(* CODESYS project Tc3_BLAKE3.library
   Company: RKe
   DefaultNamespace: Tc3_BLAKE3
   Version: 0.0.0.2
   Placeholder: Tc3_BLAKE3
   Author: Kim Robbens
   Description: Library for hash calculation with the BLAKE3 algorithm
   Title: Tc3_BLAKE3

Project tree, tasks and I/O mapping:
  libraries: Tc2_System, * (Beckhoff Automation GmbH); Tc2_Utilities, * (Beckhoff Automation GmbH); Tc3_AlgoInterfaces, * (RKe)
  DUTs/
    data type blake3_chunk_state
    data type blake3_hasher
    data type output
    data type size_t
  ITFs/
    interface IDigestBlake3: init_derive_key, init_keyed
  POUs/
    function block BLAKE3 [ST]: algorithm, chunk_state_init, chunk_state_len, chunk_state_output, chunk_state_start_flag, chunk_state_update, compress, finalize, g, hasher_add_chunk_cv, hasher_init_internal, hasher_pop_stack, hasher_push_stack, init, init_derive_key, init_keyed, key_bytes_from_hex_string, key_bytes_from_string, output_chaining_value, output_root_bytes, parent_cv, parent_output, permute, round_function, update, words_from_little_endian_bytes
  Project Information/
    function F_GetCompany [ST]
    function F_GetTitle [ST]
    function F_GetVersion [ST]
  Version/
    global variables Global_Version
  global variables ParameterList
*)

// DUTs/blake3_chunk_state
TYPE blake3_chunk_state :
STRUCT
  chaining_value				: ARRAY[0..7] OF DWORD;
  chunk_counter					: DWORD;
  block							: ARRAY[0..ParameterList.BLAKE3_BLOCK_LEN-1] OF BYTE;
  block_len						: BYTE;
  blocks_compressed				: BYTE;				
  flags							: DWORD;
END_STRUCT
END_TYPE

// DUTs/blake3_hasher
// An incremental hasher that can accept any number of writes.
TYPE blake3_hasher :
STRUCT
  chunk_state					: blake3_chunk_state;
  key_words						: ARRAY[0..7] OF DWORD;
  cv_stack 						: ARRAY[0..8*54] OF DWORD; // Space for 54 subtree chaining values:
  cv_stack_len					: BYTE;      // 2^54 * CHUNK_LEN = 2^64
  flags							: DWORD;
END_STRUCT
END_TYPE

// DUTs/output
// Each chunk or parent node can produce either an 8-word chaining value or, by
// setting the ROOT flag, any number of final output bytes. The Output struct
// captures the state just prior to choosing between those two possibilities.
TYPE output :
STRUCT
    input_chaining_value : ARRAY [0..7] OF DWORD; (* 8 x 32-bit unsigned *)
    block_words          : ARRAY [0..15] OF DWORD; (* 16 x 32-bit unsigned *)
    counter              : DWORD;  (* 64-bit unsigned integer *)
    block_len            : DWORD;  (* 32-bit unsigned integer *)
    flags                : DWORD;  (* 32-bit unsigned integer *)
END_STRUCT
END_TYPE

(*
// Each chunk or parent node can produce either an 8-word chaining value or, by
// setting the ROOT flag, any number of final output bytes. The Output struct
// captures the state just prior to choosing between those two possibilities.
typedef struct output {
  uint32_t input_chaining_value[8];
  uint32_t block_words[16];
  uint64_t counter;
  uint32_t block_len;
  uint32_t flags;
} output;
*)

// DUTs/size_t
TYPE size_t : DWORD; END_TYPE

// Version/Global_Version
{attribute 'TcGenerated'}
{attribute 'no-analysis'}
{attribute 'linkalways'}
// This function has been automatically generated from the project information.
VAR_GLOBAL CONSTANT
	{attribute 'const_non_replaced'}
	stLibVersion_Tc3_BLAKE3 : ST_LibVersion := (iMajor := 0, iMinor := 0, iBuild := 0, iRevision := 2, nFlags := 0, sVersion := '0.0.0.2');
END_VAR

// ParameterList
{attribute 'qualified_only'}
VAR_GLOBAL CONSTANT
	BLAKE3_OUT_LEN 					: DWORD := 32;
	BLAKE3_KEY_LEN 					: DWORD := 32;
	BLAKE3_BLOCK_LEN 	 			: DWORD := 64;
	BLAKE3_CHUNK_LEN  				: DWORD := 1024;

	MSG_PERMUTATION					: ARRAY[0..15] OF DWORD := [	2, 6,  3,  10, 7, 0,  4,  13,
                                     								1, 11, 12, 5,  9, 14, 15, 8];
	IV								: ARRAY[0..7] OF DWORD := [	16#6A09E667, 16#BB67AE85, 16#3C6EF372, 16#A54FF53A,
																16#510E527F, 16#9B05688C, 16#1F83D9AB, 16#5BE0CD19];
	CHUNK_START 					: DWORD := SHL(1, 0);
	CHUNK_END 						: DWORD := SHL(1, 1);
	PARENT 							: DWORD := SHL(1, 2);
	ROOT 							: DWORD := SHL(1, 3);
	KEYED_HASH 						: DWORD := SHL(1, 4);
	DERIVE_KEY_CONTEXT 				: DWORD := SHL(1, 5);
	DERIVE_KEY_MATERIAL 			: DWORD := SHL(1, 6);

END_VAR

// ITFs/IDigestBlake3
INTERFACE IDigestBlake3 EXTENDS IDigest

// Initialize the `Hasher` for the key derivation function. 
// The context string should be hardcoded, globally unique, and application-specific.
METHOD init_derive_key
VAR_INPUT CONSTANT
    context 					: STRING; // The context string
END_VAR
VAR
    context_key 				: ARRAY[0..parameterList.BLAKE3_KEY_LEN-1] 		OF BYTE; 
    context_key_words 			: ARRAY[0..(parameterList.BLAKE3_KEY_LEN/4)-1] 	OF DWORD;
END_VAR
END_METHOD

// Initialize the `Hasher` for the keyed hash function.
METHOD init_keyed
VAR_INPUT CONSTANT
    key 						: ARRAY[0..parameterList.BLAKE3_KEY_LEN-1] 		OF BYTE; 
END_VAR
VAR
    key_words 					: ARRAY[0..(parameterList.BLAKE3_KEY_LEN/4)-1] 	OF DWORD;
END_VAR
END_METHOD

END_INTERFACE

// POUs/BLAKE3
{attribute 'no_explicit_call' := 'do not call this POU directly, use the hash method'} 
FUNCTION_BLOCK BLAKE3 IMPLEMENTS IDigest
VAR
	// Hasher parameters
	self						: blake3_hasher; 					

	// Hasher assertions
	bAssertFailed				: BOOL;
END_VAR
VAR CONSTANT
	_ALGORITHM					: STRING := 'BLAKE3';
END_VAR

PROPERTY algorithm : string
GET
algorithm := _ALGORITHM;
END_GET
END_PROPERTY

METHOD PRIVATE chunk_state_init
VAR_INPUT
	self						: REFERENCE TO blake3_chunk_state;
END_VAR
VAR_INPUT CONSTANT
    key_words 					: ARRAY[0..7] OF DWORD;
    chunk_counter 				: DWORD;
    flags     					: DWORD;
END_VAR
VAR
    i 							: INT;
END_VAR
memcpy(ADR(self.chaining_value), ADR(key_words), SIZEOF(self.chaining_value));
self.chunk_counter 				:= chunk_counter;
memset(ADR(self.block), 16#0, SIZEOF(self.block));
self.block_len 					:= 0;
self.blocks_compressed 			:= 0;
self.flags 						:= flags;
END_METHOD

METHOD PRIVATE chunk_state_len : DWORD
VAR_INPUT
	self						: REFERENCE TO blake3_chunk_state;
END_VAR
chunk_state_len 		:= ParameterList.BLAKE3_BLOCK_LEN * TO_DWORD(self.blocks_compressed) + TO_DWORD(self.block_len);
END_METHOD

METHOD PRIVATE chunk_state_output : output
VAR_INPUT
	self						: REFERENCE TO blake3_chunk_state;
END_VAR
VAR
	ret_						: output;
    i 							: INT;
END_VAR
memcpy(ADR(ret_.input_chaining_value), ADR(self.chaining_value), SIZEOF(ret_.input_chaining_value));
words_from_little_endian_bytes(self.block, SIZEOF(self.block), ret_.block_words);
ret_.counter 					:= self.chunk_counter;
ret_.block_len 					:= TO_DWORD(self.block_len);
ret_.flags 						:= self.flags OR chunk_state_start_flag(self) OR ParameterList.CHUNK_END;
chunk_state_output				:= ret_;
END_METHOD

METHOD PRIVATE chunk_state_start_flag : DWORD
VAR_INPUT
	self						: REFERENCE TO blake3_chunk_state;
END_VAR
IF self.blocks_compressed = 0 THEN
    chunk_state_start_flag := ParameterList.CHUNK_START;
ELSE
    chunk_state_start_flag := 0;
END_IF
END_METHOD

METHOD PRIVATE chunk_state_update
VAR_INPUT
	self 						: REFERENCE TO blake3_chunk_state;	
END_VAR
VAR_INPUT CONSTANT
    input 						: POINTER TO BYTE; 
    input_len 					: DWORD;
END_VAR
VAR
    input_u8 					: POINTER TO BYTE;
    want, take 					: DWORD;
    i 							: DWORD;
    block_words 				: ARRAY[0..15] OF DWORD;
    out16 						: ARRAY[0..15] OF DWORD;
    temp_flag 					: DWORD;
END_VAR
input_u8						:= input;
WHILE (input_len > 0) 			DO
    // If the block buffer is full, compress it and clear it. More input is
    // coming, so this compression is not CHUNK_END.
    IF (self.block_len = parameterList.BLAKE3_BLOCK_LEN) THEN
		words_from_little_endian_bytes(self.block, parameterList.BLAKE3_BLOCK_LEN,
                                     block_words);
		compress(self.chaining_value, block_words, self.chunk_counter,
               parameterList.BLAKE3_BLOCK_LEN, self.flags OR chunk_state_start_flag(self),
               out16);
		memcpy(ADR(self.chaining_value), ADR(out16), SIZEOF(self.chaining_value));
      	self.blocks_compressed := self.blocks_compressed + 1;
      	memset(ADR(self.block), 16#0, SIZEOF(self.block));
      	self.block_len := 0;			   
	END_IF
    // Copy input bytes into the block buffer.
    want := ParameterList.BLAKE3_BLOCK_LEN - self.block_len;
    take := want;
    IF (input_len < want) 	THEN
    	take := input_len;
    END_IF
    memcpy(ADR(self.block[self.block_len]), input_u8, take);
    self.block_len 	:= self.block_len + TO_BYTE(take);
    input_u8 		:= input_u8 + TO_BYTE(take);
    input_len 		:= input_len - TO_DWORD(take);	
END_WHILE
END_METHOD

METHOD PRIVATE compress
VAR_INPUT CONSTANT
	chaining_value						: ARRAY[0..7] OF DWORD;
	block_words							: ARRAY[0..15] OF DWORD;
END_VAR
VAR_INPUT
	counter								: DWORD;
	block_len							: DWORD;
	flags								: DWORD;
	out									: REFERENCE TO ARRAY[0..15] OF DWORD;
END_VAR
VAR
	state								: ARRAY[0..15] OF DWORD;
	block								: ARRAY[0..15] OF DWORD;
	i									: INT;
END_VAR
state[00] := chaining_value[0];
state[01] := chaining_value[1];
state[02] := chaining_value[2];
state[03] := chaining_value[3];
state[04] := chaining_value[4];
state[05] := chaining_value[5];
state[06] := chaining_value[6];
state[07] := chaining_value[7];
state[08] := ParameterList.IV[0];
state[09] := ParameterList.IV[1];
state[10] := ParameterList.IV[2];
state[11] := ParameterList.IV[3];
state[12] := TO_DWORD(counter);
state[13] := 0; // TO_DWORD(SHR(counter, 32)); we don't use LWORD
state[14] := block_len;
state[15] := flags;

memcpy(ADR(block), ADR(block_words), SIZEOF(block));

round_function(state, block); // round 1
permute(block);
round_function(state, block); // round 2
permute(block);
round_function(state, block); // round 3
permute(block);
round_function(state, block); // round 4
permute(block);
round_function(state, block); // round 5
permute(block);
round_function(state, block); // round 6
permute(block);
round_function(state, block); // round 7

FOR i := 0 TO 7 DO
	state[i] := state[i] XOR state[i + 8];
	state[i + 8] := state[i + 8] XOR chaining_value[i];	
END_FOR

memcpy(ADR(out), ADR(state), SIZEOF(state));
END_METHOD

// Finalize the hash and write any number of output bytes.
METHOD finalize
(*VAR_INPUT CONSTANT
	self						: REFERENCE TO blake3_hasher;
END_VAR
VAR_INPUT
    out     					: REFERENCE TO ARRAY [0..ParameterList.BLAKE3_OUT_LEN-1] OF BYTE;
END_VAR*)
VAR_IN_OUT
    out     					: ARRAY [*] OF BYTE;
END_VAR
VAR
    current_output 				: output;
    parent_nodes_remaining   	: DWORD;
    current_cv     				: ARRAY[0..7] OF DWORD;
END_VAR
// Starting with the output from the current chunk, compute all the parent
// chaining values along the right edge of the tree, until we have the root
// output.
current_output 				:= chunk_state_output(self.chunk_state);

parent_nodes_remaining 		:= self.cv_stack_len;
WHILE (parent_nodes_remaining > 0) DO
	parent_nodes_remaining	:= parent_nodes_remaining - 1;
    output_chaining_value(current_output, current_cv);
	current_output 			:= parent_output(ADR(self.cv_stack[parent_nodes_remaining * 8]), current_cv, self.key_words, self.flags);
END_WHILE

// Output the root output.
output_root_bytes(current_output, out);
END_METHOD

// The mixing function, G, which mixes either a column or a diagonal.
METHOD PRIVATE g
VAR_INPUT
	state 					: REFERENCE TO ARRAY[0..15] OF DWORD;	
	a, b, c, d 				: DWORD;
	mx, my 					: DWORD;
END_VAR
state[a] := state[a] + state[b] + mx;
state[d] := ROR((state[d] XOR state[a]), 16);
state[c] := state[c] + state[d];
state[b] := ROR((state[b] XOR state[c]), 12);
state[a] := state[a] + state[b] + my;
state[d] := ROR((state[d] XOR state[a]), 8);
state[c] := state[c] + state[d];
state[b] := ROR((state[b] XOR state[c]), 7);
END_METHOD

// Section 5.1.2 of the BLAKE3 spec explains this algorithm in more detail.
METHOD PRIVATE hasher_add_chunk_cv
VAR_INPUT
	self						: REFERENCE TO blake3_hasher;
	new_cv						: REFERENCE TO ARRAY[0..7] OF DWORD;
	total_chunks				: DWORD;
END_VAR
// This chunk might complete some subtrees. For each completed subtree, its
// left child will be the current top entry in the CV stack, and its right
// child will be the current value of `new_cv`. Pop each left child off the
// stack, merge it with `new_cv`, and overwrite `new_cv` with the result.
// After all these merges, push the final value of `new_cv` onto the stack.
// The number of completed subtrees is given by the number of trailing 0-bits
// in the new total number of chunks.
WHILE ((total_chunks AND 1) = 0) DO
	parent_cv(hasher_pop_stack(), new_cv, self.key_words, self.flags, new_cv);
	total_chunks := SHR(total_chunks, 1);
END_WHILE
hasher_push_stack(new_cv);
END_METHOD

METHOD PRIVATE hasher_init_internal
VAR_INPUT CONSTANT
    key_words 					: ARRAY[0..7] OF DWORD;
    flags     					: DWORD;
END_VAR
chunk_state_init(self.chunk_state, key_words, 0, flags);
memcpy(ADR(self.key_words), ADR(key_words), SIZEOF(key_words));
self.cv_stack_len 		:= 0;
self.flags 				:= flags;
END_METHOD

// Returns a pointer to the popped CV, which is valid until the next push.
METHOD PRIVATE hasher_pop_stack : POINTER TO ARRAY[0..7] OF DWORD
VAR
    idx 						: DWORD;
END_VAR
self.cv_stack_len := self.cv_stack_len - 1;
hasher_pop_stack := adr(self.cv_stack[self.cv_stack_len * 8]);
END_METHOD

METHOD PRIVATE hasher_push_stack
VAR_INPUT
    cv 							: ARRAY[0..7] OF DWORD;
END_VAR
VAR
    i 							: INT;
    destIndex 					: DWORD;
END_VAR
memcpy(ADR(self.cv_stack[self.cv_stack_len * 8]), ADR(cv), 8 * 4);
self.cv_stack_len := self.cv_stack_len + 1;
END_METHOD

// Initialize the `Hasher` for a regular hash function
METHOD init
hasher_init_internal(ParameterList.IV, 0);
END_METHOD

// Initialize the `Hasher` for the key derivation function. 
// The context string should be hardcoded, globally unique, and application-specific.
METHOD init_derive_key
VAR_INPUT CONSTANT
    context 					: STRING; // The context string
END_VAR
VAR
    context_key 				: ARRAY[0..parameterList.BLAKE3_KEY_LEN-1] 		OF BYTE; 
    context_key_words 			: ARRAY[0..(parameterList.BLAKE3_KEY_LEN/4)-1] 	OF DWORD;
END_VAR
hasher_init_internal(ParameterList.IV, ParameterList.DERIVE_KEY_CONTEXT);
update(ADR(context), len2(ADR(context)));
finalize(context_key);
words_from_little_endian_bytes(context_key, parameterList.BLAKE3_KEY_LEN, context_key_words);
hasher_init_internal(context_key_words, ParameterList.DERIVE_KEY_MATERIAL);
END_METHOD

// Initialize the `Hasher` for the keyed hash function.
METHOD init_keyed
VAR_INPUT CONSTANT
    key 						: ARRAY[0..parameterList.BLAKE3_KEY_LEN-1] 		OF BYTE; 
END_VAR
VAR
    key_words 					: ARRAY[0..(parameterList.BLAKE3_KEY_LEN/4)-1] 	OF DWORD;
END_VAR
words_from_little_endian_bytes(key, parameterList.BLAKE3_KEY_LEN, key_words);
hasher_init_internal(key_words, ParameterList.KEYED_HASH);
END_METHOD

// convert a string representing hex byte to a hex byte array 
METHOD PUBLIC key_bytes_from_hex_string
VAR_INPUT CONSTANT
	hex_key						: REFERENCE TO STRING;
END_VAR
VAR_IN_OUT
	out							: ARRAY[*] OF BYTE;
END_VAR
VAR
    base_idx 					: POINTER TO STRING(1);
    input_idx 					: POINTER TO STRING(1);
	nibbleH						: STRING(1);	
	nibbleL						: STRING(1);	
	i							: DWORD;
END_VAR
base_idx := ADR(hex_key);
FOR i := 0 TO TO_DWORD(UPPER_BOUND(out, 1)) DO
	input_idx := base_idx + 2*i;
	nibbleH := input_idx^;
	out[i] := HEXCHRNIBBLE_TO_BYTE(nibbleH);
	input_idx := base_idx + 2*i + 1;
	nibbleL := input_idx^;
	out[i] := SHL(out[i],4) + HEXCHRNIBBLE_TO_BYTE(nibbleL);
END_FOR
END_METHOD

// convert a string to a hex byte array 
METHOD PUBLIC key_bytes_from_string
VAR_INPUT CONSTANT
	key							: REFERENCE TO STRING;	
END_VAR
VAR_IN_OUT
	out							: ARRAY[*] OF BYTE;
END_VAR
VAR
	temp 						: ARRAY[0..MAX_STRING_LENGTH] OF BYTE;
	length						: DWORD;
END_VAR
temp 	:= MAXSTRING_TO_BYTEARR(key);
length 	:= TO_DWORD(UPPER_BOUND(out, 1) - LOWER_BOUND(out, 1)); 
memcpy(out, ADR(temp), length);
END_METHOD

METHOD PRIVATE output_chaining_value 
VAR_INPUT
    self 						: REFERENCE TO output; 					
    out 						: REFERENCE TO ARRAY[0..7] OF DWORD;
END_VAR
VAR
    out16 						: ARRAY[0..15] OF DWORD;
    i 							: INT;
END_VAR
// Call the compress function (must be implemented elsewhere)
compress(self.input_chaining_value, self.block_words, self.counter,
    self.block_len, self.flags,
    out16
);

// Copy first 8 DWORDs from out16 to out 
memcpy(ADR(out), ADR(out16), 8*4);
END_METHOD

METHOD PRIVATE output_root_bytes 
VAR_INPUT
    self 					: REFERENCE TO output; 
END_VAR
VAR_IN_OUT
    out 					: ARRAY[*] OF BYTE; 
END_VAR
VAR
    out_len 				: DWORD;
    out_idx 				: DWORD := 0;
	out_idxUL				: DWORD := 0;
    output_block_counter 	: DWORD := 0;
    words 					: ARRAY[0..15] OF DWORD;
    word_ 					: INT;
    byte_ 					: INT;
    temp_byte 				: BYTE;
END_VAR
out_idx		:= TO_DWORD(LOWER_BOUND(out,1));
out_idxUL	:= TO_DWORD(UPPER_BOUND(out,1));
out_len		:= out_idxUL - out_idx + 1;
WHILE out_len > 0 DO
	compress(self.input_chaining_value, self.block_words, output_block_counter,
		   self.block_len, self.flags OR self.flags OR ParameterList.ROOT, words);
    FOR word_ := 0 TO 15 DO
        FOR byte_ := 0 TO 3 DO
            IF out_len = 0 OR out_idx > out_idxUL THEN
                RETURN;
            END_IF
            temp_byte := TO_BYTE(SHR(words[word_], (8 * byte_)));
            out[out_idx] := temp_byte;
            out_idx := out_idx + 1;
            out_len := out_len - 1;
        END_FOR
    END_FOR
    output_block_counter := output_block_counter + 1;
END_WHILE
END_METHOD

METHOD PRIVATE parent_cv
VAR_INPUT CONSTANT
    left_child_cv  				: POINTER TO ARRAY[0..7] OF DWORD;
    right_child_cv 				: ARRAY[0..7] OF DWORD;
    key_words      				: ARRAY[0..7] OF DWORD;
END_VAR
VAR_INPUT
    flags          				: DWORD;
	out 						: REFERENCE TO ARRAY[0..7] OF DWORD;
END_VAR
VAR
	o							: output;
END_VAR
o := parent_output(left_child_cv, right_child_cv, key_words, flags);
// We only write to `out` after we've read the inputs. That makes it safe for
// `out` to alias an input, which we do below.
output_chaining_value(o, out);
END_METHOD

METHOD PRIVATE parent_output : output
VAR_INPUT CONSTANT
    left_child_cv  				: POINTER TO ARRAY[0..7] OF DWORD;
    right_child_cv 				: ARRAY[0..7] OF DWORD;
    key_words      				: ARRAY[0..7] OF DWORD;
END_VAR
VAR_INPUT
    flags          				: DWORD;
END_VAR
VAR
	ret_						: output;
END_VAR
memcpy(ADR(ret_.input_chaining_value), ADR(key_words), SIZEOF(ret_.input_chaining_value));
memcpy(ADR(ret_.block_words[0]), left_child_cv, 8 * 4);
memcpy(ADR(ret_.block_words[8]), ADR(right_child_cv), 8 * 4);
ret_.counter := 0; // Always 0 for parent nodes.
ret_.block_len := parameterList.BLAKE3_BLOCK_LEN; // Always BLAKE3_BLOCK_LEN (64) for parent nodes.
ret_.flags := ParameterList.PARENT OR flags;
parent_output := ret_;
END_METHOD

METHOD PRIVATE permute
VAR_INPUT
	m 						: REFERENCE TO ARRAY[0..15] OF DWORD;
END_VAR
VAR
	i						: INT;
	permuted				: ARRAY[0..15] OF DWORD;
END_VAR
FOR i := 0 TO 15 DO
	permuted[i] := m[ParameterList.MSG_PERMUTATION[i]];
END_FOR
memcpy(ADR(m), ADR(permuted), SIZEOF(permuted));
END_METHOD

METHOD PRIVATE round_function
VAR_INPUT
	state 					: REFERENCE TO ARRAY[0..15] OF DWORD;
	m 						: ARRAY[0..15] OF DWORD;
END_VAR
// Mix the columns.
g(state, 0, 4, 8, 12, m[0], m[1]);
g(state, 1, 5, 9, 13, m[2], m[3]);
g(state, 2, 6, 10, 14, m[4], m[5]);
g(state, 3, 7, 11, 15, m[6], m[7]);
// Mix the diagonals.
g(state, 0, 5, 10, 15, m[8], m[9]);
g(state, 1, 6, 11, 12, m[10], m[11]);
g(state, 2, 7, 8, 13, m[12], m[13]);
g(state, 3, 4, 9, 14, m[14], m[15]);
END_METHOD

// Add input to the hash state. This can be called any number of times.
METHOD update
VAR_INPUT
    input 						: POINTER TO BYTE; 
    input_len 					: DWORD;
END_VAR
VAR
    input_idx 					: DWORD := 0;
    want, take 					: DWORD;
    chunk_output 				: output;
    chunk_cv 					: ARRAY[0..7] OF DWORD;
    total_chunks 				: DWORD;
END_VAR
WHILE input_len > 0 DO
    // If the current chunk is complete, finalize it and reset the chunk state.
	// More input is coming, so this chunk is not ROOT.
    IF chunk_state_len(self.chunk_state) = parameterList.BLAKE3_CHUNK_LEN THEN
        chunk_output := chunk_state_output(self.chunk_state);
        output_chaining_value(chunk_output, chunk_cv);
        total_chunks := self.chunk_state.chunk_counter + 1;
        hasher_add_chunk_cv(self, chunk_cv, total_chunks);
        chunk_state_init(self.chunk_state, self.key_words, total_chunks, self.flags);
    END_IF

    // Compress input bytes into the current chunk state.
    want := parameterList.BLAKE3_CHUNK_LEN - chunk_state_len(self.chunk_state);
    take := want;
    IF input_len < want THEN
        take := input_len;
    END_IF

    chunk_state_update(self.chunk_state, ADR(input[input_idx]), take);
    input_idx := input_idx + take;
    input_len := input_len - take;
END_WHILE
END_METHOD

METHOD PRIVATE words_from_little_endian_bytes : BOOL
VAR_IN_OUT
	bytes         			: ARRAY[*] OF BYTE;   	// input ARRAY
END_VAR
VAR_INPUT
	bytes_len    	 		: DWORD;        			// length OF bytes, must be multiple OF 4
END_VAR
VAR_IN_OUT
	out           			: ARRAY[*] OF DWORD;  	// output ARRAY
END_VAR
VAR
    i 						: DWORD;
END_VAR
(*
	Endianness is the byte order used to represent multi-byte values. Little-endian means the least significant byte comes first.
	Cryptographic algorithms like BLAKE3 often work on 32-bit or 64-bit "words," but input keys and data are typically provided as byte arrays.
	For cross-platform compatibility, and to match the algorithm’s specification, you must explicitly assemble 32-bit words from bytes in little-endian order. This ensures that the hash function produces the same result on all platforms, regardless of the system's native endianness.
*)
// Assert: bytes_len must be a multiple of 4
IF (bytes_len MOD 4) <> 0 THEN
    // Set assertion failure
    bAssertFailed := TRUE;
    RETURN;
END_IF;

// Actual conversion
FOR i := 0 TO (bytes_len / 4) - 1 DO
    out[i] := TO_DWORD(bytes[4*i]) +
              SHL(TO_DWORD(bytes[4*i + 1]), 8) +
              SHL(TO_DWORD(bytes[4*i + 2]), 16) +
              SHL(TO_DWORD(bytes[4*i + 3]), 24);
END_FOR
END_METHOD

END_FUNCTION_BLOCK

// Project Information/F_GetCompany
// This function has been automatically generated from the project information.
{attribute 'signature_flag' := '1073741824'}
{attribute 'TcGenerated'}
{attribute 'no-analysis'}
FUNCTION F_GetCompany : WSTRING
VAR_INPUT
	
END_VAR

F_GetCompany := "RKe";

END_FUNCTION

// Project Information/F_GetTitle
// This function has been automatically generated from the project information.
{attribute 'signature_flag' := '1073741824'}
{attribute 'TcGenerated'}
{attribute 'no-analysis'}
FUNCTION F_GetTitle : WSTRING
VAR_INPUT
	
END_VAR

F_GetTitle := "Tc3_BLAKE3";

END_FUNCTION

// Project Information/F_GetVersion
// This function has been automatically generated from the project information.
{attribute 'signature_flag' := '1073741824'}
{attribute 'TcGenerated'}
{attribute 'no-analysis'}
FUNCTION F_GetVersion : ST_LibVersion
VAR_INPUT
	
END_VAR

F_GetVersion.iMajor := 0;
F_GetVersion.iMinor := 0;
F_GetVersion.iBuild := 0;
F_GetVersion.iRevision := 2;
F_GetVersion.sVersion := '0.0.0.2';
F_GetVersion.nFlags := 0;

END_FUNCTION
